Staubli VAL3: CommType.pjx

--- CommType.pjx ---
Parameters version=s7.8.1 stackSize=5000 millimeterUnit=true
Program file=start.pgx
Program file=stop.pgx
Data file=CommType.dtx

--- CommType.dtx ---
public num INVALID
public num TOPIC
public num SERVICE_REQUEST
public num SERVICE_REPLY
